(* IEC 61131-3 sources: plcassist-cli/packages/volt-lsp-iec/test-corpus/pro2193/Device/Plc Logic/Application/99 Library/Function Blocks/Actuators/Vacuums, 4 files *)

(* ---- VacuumFB.fb ---- *)
// Control a vacuum output; vacuum high level is not measured!
{attribute 'symbol' := 'none'}
FUNCTION_BLOCK PUBLIC VacuumFB
EXTENDS ActuatorWithManualControlAndAlarm_BaseFB
IMPLEMENTS IVacuum
VAR_INPUT
	refVacuumHighTime		: REFERENCE TO REAL;	// Optional: vacuum is high after this timeout
	refReleaseVacuumTime	: REFERENCE TO REAL;	// Optional: vacuum is released after this timeout
	enableDuringSemiAuto	: BOOL := FALSE;
END_VAR
VAR
	{attribute 'symbol' := 'read'}	Output					: ActuatorFB;
	VacuumHighTimer			: BTON;
	ReleaseVacuumTimer		: BTON;
END_VAR

SUPER^();

// Instantiate the output
Output();

SetVacuumHighTimer();

ReleaseVacuumTimer.Set(
			In := NOT IsTurnedOn,
			Pt := SEL(__ISVALIDREF(refReleaseVacuumTime), 0, refReleaseVacuumTime));

END_FUNCTION_BLOCK

METHOD PROTECTED Alarms
END_METHOD

METHOD PROTECTED ManualControl
VAR_INPUT
	minButtonPushed			: BOOL;		// Both the software button (on screen) and the hardware button (if attached)
	plusButtonPushed		: BOOL;		// Both the software button (on screen) and the hardware button (if attached)
END_VAR
IF plusButtonPushed THEN
	Set();
END_IF

IF minButtonPushed THEN
	Reset();
END_IF
END_METHOD

// Maps the actuator to the physical output
METHOD Map : BOOL
// Disabe mapping when machine is running without vacuums
IF SER.OperationMode = SER_OperationModeType.SemiAuto
AND HMI.SemiAutoMode = enumSemiAutoModeType.WithoutVacuums
AND NOT enableDuringSemiAuto
THEN
	Map := FALSE;
ELSE
	Map := Output.Map();
END_IF
END_METHOD

// Release (resets) the vacuum output. Returns true after a timer.
METHOD Release : BOOL
VAR_INPUT
END_VAR
Reset();

Release	:= ReleaseVacuumTimer.Q;
END_METHOD

// Reset the output (=False)
METHOD Reset
Output.Reset();
END_METHOD

// Set the output (=True)
METHOD Set : BOOL
Output.Set();

Set := IsHigh;
END_METHOD

// Set the output True or False
METHOD SetOrReset
VAR_INPUT
	xValue	: BOOL;
END_VAR
Output.SetOrReset(xValue);
END_METHOD

METHOD PROTECTED SetVacuumHighTimer
VAR_INPUT
END_VAR
VacuumHighTimer.Set(
			In := IsTurnedOn,
			Pt := SEL(__ISVALIDREF(refVacuumHighTime), 0, refVacuumHighTime));
END_METHOD

// Vacuum input is high (after optional timer)
{attribute 'monitoring':='call'}
PROPERTY IsHigh : BOOL
GET
VAR
END_VAR
IsHigh	:= VacuumHighTimer.Q;
END_GET
END_PROPERTY

// Get state of the output (Normally you could call Map(), but with vacuums the Map() method may return false if machine runs without vacuums.
{attribute 'monitoring':='call'}
PROPERTY IsTurnedOn : BOOL
GET
VAR
END_VAR
IsTurnedOn	:= Output.Map();
END_GET
END_PROPERTY

(* ---- VacuumWithInputFB.fb ---- *)
// Control a vacuum output and measure the vacuum level
{attribute 'symbol' := 'none'}
FUNCTION_BLOCK PUBLIC VacuumWithInputFB
EXTENDS VacuumFB
IMPLEMENTS IVacuum
VAR_INPUT
	{attribute 'symbol' := 'read'}	input1					: BOOL;				// Input 1 of Vacuum sensor (Vacuum level reached)
	errorId					: WORD;
END_VAR
VAR
	{attribute 'symbol' := 'read'}	vacuumHighDuration		: REAL;				// The amount of time elapsed before vacuum level reached.
	NoVacuumAlarm			: SetErrorFB;
	MeasureMaxTime			: StopwatchFB;
	vacuumState				: USINT;
END_VAR

SUPER^();

// Onderstaand is een idee van Arnoud
// Verschil detecteren tussen: No vacuum, en Vacuum lost
// Hier 2 verschillende alarmmeldingen van maken...

IF NOT Map() THEN
	vacuumState					:= 0;
ELSE
	CASE vacuumState OF
		0:	// vacuum off
			IF Map() THEN
				vacuumState		:= 1;
			END_IF
		1:	// vacuum on
			IF input1 THEN
				vacuumState		:= 2;
			END_IF
		2:	// vacuum detected
			IF NOT input1 THEN
				vacuumState		:= 3;
			END_IF
		3:	// vacuum lost
			;
	END_CASE
END_IF

END_FUNCTION_BLOCK

METHOD PROTECTED Alarms

// Remember that this method may be replaced by another when deriving from this base FB.
NoVacuumAlarm(
	moduleHandler	:= moduleHandler,
	textRefId		:= textRefId,
	alarmCondition	:= alarmEnable AND (input1 XOR Output.Map()) AND errorId <> 0,
	alarmDelay		:= alarmDelay,
	errorId			:= errorId,
	severity		:= severity,
	reaction		:= reaction,
	active			=> );

IF alarmEnable AND Output.Map() AND NOT input1 AND errorId <> 0 THEN
	vacuumHighDuration	:= NoVacuumAlarm.ElapsedTime;
END_IF

MeasureMaxTime.Monitor(
	in				:= Output.Map() AND NOT input1);
END_METHOD

METHOD PUBLIC SetMonitoring
VAR_INPUT
	itfAddLog		: EdgePcLogging.IAddLog;
	plcDataType		: PlcDataType;
END_VAR
MeasureMaxTime.SetMonitoring(itfAddLog, plcDataType);
END_METHOD

METHOD PROTECTED SetVacuumHighTimer
VAR_INPUT
END_VAR
VacuumHighTimer.Set(
			In := input1,
			Pt := SEL(__ISVALIDREF(refVacuumHighTime), 0, refVacuumHighTime));
END_METHOD

(* ---- VacuumWithPressureFB.fb ---- *)
// Control a vacuum output and measure the vacuum level. Use the second input to measure the pressure (check if a label is present)
{attribute 'symbol' := 'none'}
FUNCTION_BLOCK FINAL VacuumWithPressureFB
EXTENDS VacuumWithInputFB
IMPLEMENTS IVacuum
VAR_INPUT
	{attribute 'symbol' := 'read'}	input2					: BOOL;				// Input 2 of Vacuum sensor (Pressure level reached)
END_VAR

SUPER^();

END_FUNCTION_BLOCK

{attribute 'monitoring':='call'}
PROPERTY HasPressure : BOOL
GET
VAR
END_VAR
HasPressure := input2;
END_GET
END_PROPERTY

(* ---- VacuumWithTwoInputsFB.fb ---- *)
// Control a vacuum output and measure the vacuum level. Vacuum high is determent by 2 separate inputs
{attribute 'symbol' := 'none'}
FUNCTION_BLOCK FINAL VacuumWithTwoInputsFB
EXTENDS VacuumWithInputFB
IMPLEMENTS IVacuum
VAR_INPUT
	{attribute 'symbol' := 'read'}	input2					: BOOL;				// Second vacuum sensor
END_VAR

SUPER^();

END_FUNCTION_BLOCK

METHOD PROTECTED Alarms

// This method wil override the original method in the base FB
NoVacuumAlarm(
	moduleHandler	:= moduleHandler,
	textRefId		:= textRefId,
	alarmCondition	:= alarmEnable AND ((input1 AND input2) XOR Output.Map()) AND errorId <> 0,
	alarmDelay		:= alarmDelay,
	errorId			:= errorId,
	severity		:= severity,
	reaction		:= reaction,
	active			=> );

IF alarmEnable AND Output.Map() AND (NOT input1 OR NOT input2) AND errorId <> 0 THEN
	vacuumHighDuration	:= NoVacuumAlarm.ElapsedTime;
END_IF

MeasureMaxTime.Monitor(
	in				:= Output.Map() AND (NOT input1 OR NOT input2));
END_METHOD

METHOD PROTECTED SetVacuumHighTimer
VAR_INPUT
END_VAR
VacuumHighTimer.Set(
			In := input1 AND input2,
			Pt := SEL(__ISVALIDREF(refVacuumHighTime), 0, refVacuumHighTime));
END_METHOD
